
// ===== library: MasterCopy "udt_gw_alive_timer" =====

TYPE "udt_gw_alive_timer"
   STRUCT
      Ton : Array[0..2] of TON_TIME;
      Tp_send : TP_TIME;
   END_STRUCT;
END_TYPE

// ===== library: MasterCopy "Copy of Program blocks in gw_alive_system" =====

// folder: gw_alive_system

DATA_BLOCK "db_gw_alive_system"   // DB910
{ S7_Optimized_Access := 'TRUE' }
VERSION : 0.1
   VAR
      alive_fault : Bool;
      alive_receive : Bool;
      alive_send : Bool;
   END_VAR
BEGIN
END_DATA_BLOCK

FUNCTION_BLOCK "fb_gw_alive_system"   // FB910, FBD
{ S7_Optimized_Access := 'TRUE' }
VERSION : 0.1
   VAR
      timer_recovery : "udt_gw_alive_timer";
   END_VAR
BEGIN

REGION Network 1: check system alive
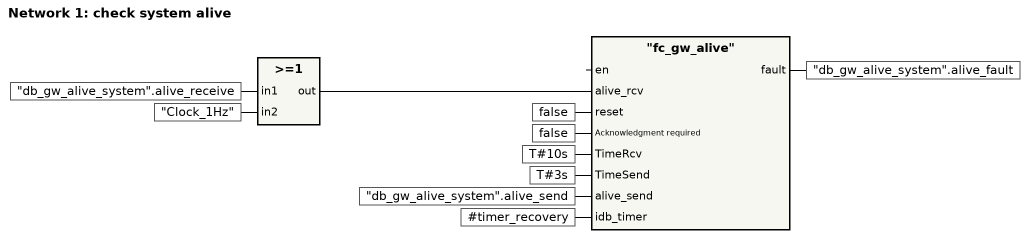
   "fc_gw_alive"(alive_rcv := "db_gw_alive_system".alive_receive OR "Clock_1Hz",
                 reset := false,
                 "Acknowledgment required" := false,
                 TimeRcv := T#10s,
                 TimeSend := T#3s,
                 alive_send := "db_gw_alive_system".alive_send,
                 idb_timer := #timer_recovery,
                 fault => "db_gw_alive_system".alive_fault);
END_REGION
END_FUNCTION_BLOCK

FUNCTION "fc_gw_alive" : Void   // FC910, FBD
{ S7_Optimized_Access := 'TRUE' }
VERSION : 0.1
   VAR_INPUT
      alive_rcv : Bool;
      reset : Bool;
      "Acknowledgment required" : Bool;
      TimeRcv : Time;
      TimeSend : Time;
   END_VAR
   VAR_OUTPUT
      fault : Bool;
   END_VAR
   VAR_IN_OUT
      alive_send : Bool;
      idb_timer : "udt_gw_alive_timer";
   END_VAR
   VAR_TEMP
      ton_dn : Bool;
      toff_dn : Bool;
      quitt : Bool;
   END_VAR
BEGIN

REGION Network 1: Alive On Timer
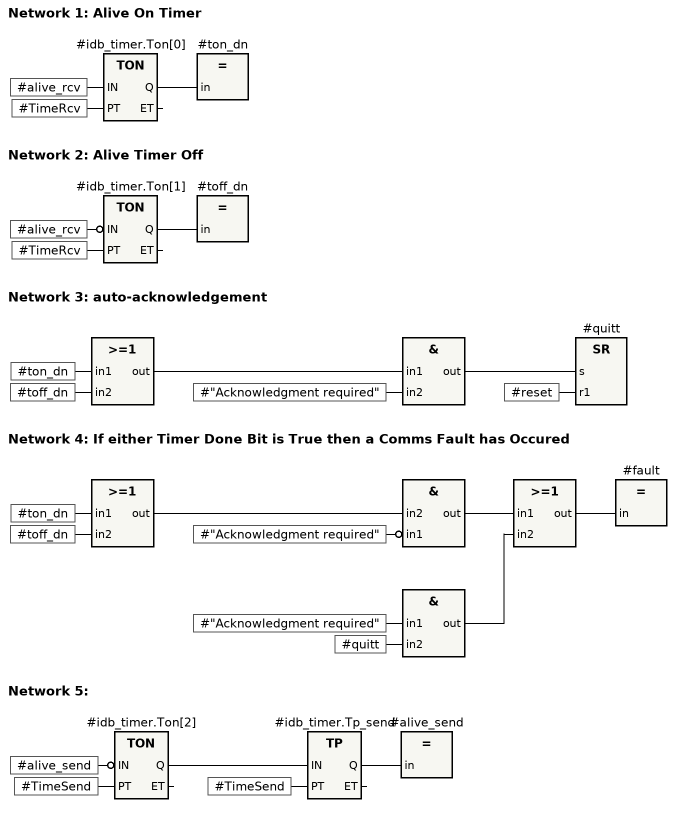
   #idb_timer.Ton[0].TON(IN := #alive_rcv, PT := #TimeRcv);
   #ton_dn := #idb_timer.Ton[0].Q;
END_REGION

REGION Network 2: Alive Timer Off
   #idb_timer.Ton[1].TON(IN := NOT #alive_rcv, PT := #TimeRcv);
   #toff_dn := #idb_timer.Ton[1].Q;
END_REGION

REGION Network 3: auto-acknowledgement
   IF (#ton_dn OR #toff_dn) AND #"Acknowledgment required" THEN
       #quitt := TRUE;   // SR flip-flop
   END_IF;
   IF #reset THEN #quitt := FALSE; END_IF;
END_REGION

REGION Network 4: If either Timer Done Bit is True then a Comms Fault has Occured
   #fault := ((#ton_dn OR #toff_dn) AND NOT #"Acknowledgment required") OR (#"Acknowledgment required" AND #quitt);
END_REGION

REGION Network 5
   #idb_timer.Ton[2].TON(IN := NOT #alive_send, PT := #TimeSend);
   #idb_timer.Tp_send.TP(IN := #idb_timer.Ton[2].Q, PT := #TimeSend);
   #alive_send := #idb_timer.Tp_send.Q;
END_REGION
END_FUNCTION